// TwinCAT 3 PLC project PlcOpen_Test
// ProgramVersion: 3.1.4024.0
// libraries:
//   Tc2_Standard, * (Beckhoff Automation GmbH)
//   Tc2_System, * (Beckhoff Automation GmbH)
//   Tc2_Utilities, * (Beckhoff Automation GmbH)
//   Tc3_Module, * (Beckhoff Automation GmbH)
//   Tc3_PLCopen_OpcUa, * (Beckhoff Automation GmbH)
//   Tc2_OpcUa,3.3.2.0,Beckhoff Automation GmbH
// project tree:
//   DUTs/01_Strukturen/ SystemControlWord.TcDUT, SystemStatusWord.TcDUT
//   / GlobalTextList.TcGTLO, PlcTask.TcTTO, Visualisierungsmanager.TcVMO (not stored), VISU_TASK.TcTTO
//   GVLs/ GVL.TcGVL
//   POUs/01_Funktionsblock/ FB_Kommunikation.TcPOU
//   POUs/ Anlage.TcPOU, MAIN.TcPOU
//   VISUs/ Test_Visu.TcVIS
// real-time tasks:
//   TASK PlcTask: cycle T#10ms, priority 20, ADS port 350
//   TASK VISU_TASK: cycle T#200000us, priority 30, ADS port 351

CONFIGURATION PlcOpen_Test
    RESOURCE PLC ON TwinCAT3
        TASK PlcTask(INTERVAL := T#10ms, PRIORITY := 20);
        TASK VISU_TASK(INTERVAL := T#200000us, PRIORITY := 30);
        PROGRAM MAIN WITH PlcTask : MAIN;
        PROGRAM VisuElems_Visu_Prg WITH VISU_TASK : VisuElems.Visu_Prg;
    END_RESOURCE
END_CONFIGURATION

// ---- DUTs/01_Strukturen/SystemControlWord.TcDUT
TYPE SystemControlWord :
STRUCT			
	PowerOn			:BOOL;			// Einschalten von Reaktoreinheit
	SekReakt		:INT;			// Definierter sekundär-Reaktor
	Leitung			:INT;			// Definiert welche Leitung verwendet wird
	Temp			:REAL;			// Definierte Temperatur für Heiz- / Kühlprozess
	Enlteermenge	:REAL;			// Zu entleerende Menge
	Pumpmenge		:REAL;			// Zu pumpende Menge
	Haltedauer		:TIME;			// Wie lange soll TEmperatur gehalten werden
	Ruehrdauer		:TIME;			// Wie lange soll gerührt werden 
	Wartedauer		:TIME;			// Wie lange soll gerührt werden
	Zirkulierdauer	:TIME;			// Wie lange soll zirkuliert werden
END_STRUCT
END_TYPE

// ---- DUTs/01_Strukturen/SystemStatusWord.TcDUT
TYPE SystemStatusWord :
STRUCT
	SysReady		:BOOL;		// System ist eingeschalten und bereit
	PrimReady		:BOOL;		// Primärreaktor ist bereit für den Prozess
	PrimActiv		:BOOL;		// Primärreaktor führt Prozess aus
	SekReady		:BOOL;		// Sekundärreaktor ist bereit für den Prozess
	SekActiv		:BOOL;		// Sekundärreaktor führt Prozess aus
	GF1Activ		:BOOL;		// Heiz- / Kühlprozess läuft
	GF2Activ		:BOOL;		// Entleerprozess läuft
	GF3Activ		:BOOL;		// Pumpprozess läuft
	GF4Activ		:BOOL;		// Halteprozess läuft
	GF5Activ		:BOOL;		// Rührprozess läuft
	GF6Activ		:BOOL;		// Warteprozess läuft
	GF7Activ		:BOOL;		// Auffüllprozess läuft
	GF8Activ		:BOOL;		// Zirkulierprozess läuft
END_STRUCT
END_TYPE

// ---- GVLs/GVL.TcGVL
{attribute 'qualified_only'}
VAR_GLOBAL
	IP			:STRING(MAX_STRING_LENGTH) := 'opc.tcp://169.254.240.2:4840';
	NameSpace	:STRING(MAX_STRING_LENGTH) := 'urn:BeckhoffAutomation:Ua:PLC1';
	
	SW		:SystemStatusWord;
	CW		:SystemControlWord;
END_VAR

// ---- POUs/MAIN.TcPOU
PROGRAM MAIN
VAR
	Check			:BOOL;
END_VAR

Anlage();

END_PROGRAM

// ---- POUs/Anlage.TcPOU
PROGRAM Anlage
VAR
	Kom_Reaktor_1		:FB_Kommunikation;
	
END_VAR

Kom_Reaktor_1(I_sIP := GVL.IP, SW := GVL.SW); // FB_Kommunikation
GVL.CW := Kom_Reaktor_1.CW;

END_PROGRAM

// ---- POUs/01_Funktionsblock/FB_Kommunikation.TcPOU
FUNCTION_BLOCK FB_Kommunikation
VAR_INPUT
	I_sIP		:STRING;
	SW			:SystemStatusWord;
END_VAR

VAR_OUTPUT
	CW			:SystemControlWord;
	Busy		:BOOL;
	Error		:BOOL;
	ErrorID		:DWORD;
END_VAR

VAR
	Connect				:UA_Connect;
	Disconnect			:UA_Disconnect; 
	Read 				:UA_Read;
	Write				:UA_Write;
	Node				:UA_NodeGetHandle;
	NameSpaceIndex		:UA_GetNamespaceIndex;
	
	ConnectInfo			:ST_UASessionConnectInfo;
	NodeID				:ST_UANodeID;
	NodeInfo			:ST_UANodeAdditionalInfo;
	
	ConnectionHdl		:DWORD;
	NoteHdl				:DWORD;
	NameSpace			:UINT;
	IndexRangeCount		:UINT := 1;
	IndexRange			:ARRAY [1..nMaxIndexRange] OF ST_UAIndexRange;
	NodeIdentifier		:STRING(MAX_STRING_LENGTH) := 'GVL_OPC_UA.SW';
	ReadData			:SystemStatusWord; 		// change to node data type
END_VAR

// Definition der Verbindungsinformationen
ConnectInfo.tSessionTimeout := T#1M;
ConnectInfo.tConnectTimeout := T#1M;
ConnectInfo.sApplicationName := '';
ConnectInfo.eSecurityMode := eUASecurityMsgMode_Sign_Encrypt;				// 3 = Sign_Encrypted
ConnectInfo.eSecurityPolicyUri := eUASecurityPolicy_Basic256Sha256;			// 4 = Basic256  
ConnectInfo.eTransportProfileUri := eUATransportProfileUri_UATcp;			// 1 = UATcp
ConnectInfo.stUserIdentTokenType.eUserIdentTokenType := eUAUITT_Username;	// 1 = Username
ConnectInfo.stUserIdentTokenType.sTokenParam1 := 'Administrator';			// Username
ConnectInfo.stUserIdentTokenType.sTokenParam2 := '1';						// PW

GVL.SW := ReadData;

ACTION ACT_Connect:
Connect(ServerUrl := I_sIP, SessionConnectInfo := ConnectInfo, Timeout := T#5s); // UA_Connect
Busy := Connect.Busy;
ConnectionHdl := Connect.ConnectionHdl;
Error := Connect.Error;
ErrorID := Connect.ErrorID;
END_ACTION

ACTION ACT_Disconnect:
Busy := Disconnect.Busy;
Error := Disconnect.Error;
ErrorID := Disconnect.ErrorID;
Disconnect(ConnectionHdl := ConnectionHdl, Timeout := T#5s); // UA_Disconnect
END_ACTION

ACTION ACT_GetNameSpaceIndex:
Busy := NameSpaceIndex.Busy;
Error := NameSpaceIndex.Error;
ErrorID := NameSpaceIndex.ErrorID;
NameSpaceIndex(ConnectionHdl := ConnectionHdl, NamespaceUri := GVL.NameSpace, Timeout := T#5s); // UA_GetNamespaceIndex
NameSpace := NameSpaceIndex.NamespaceIndex;
END_ACTION

ACTION ACT_GetNodes:
NoteHdl := Node.NodeHdl;
Busy := Node.Busy;
Error := Node.Error;
ErrorID := Node.ErrorID;
Node(ConnectionHdl := ConnectionHdl, NodeID := NodeID, Timeout := T#5s); // UA_NodeGetHandle
END_ACTION

ACTION ACT_Read:
Busy := Read.Busy;
Error := Read.Error;
ErrorID := Read.ErrorID;
Read(
    ConnectionHdl := ConnectionHdl,
    NodeHdl := NoteHdl,
    stNodeAddInfo := NodeInfo,
    pVariable := ADR(ReadData),
    cbData := SIZEOF(ReadData),
    Timeout := T#5s); // UA_Read
END_ACTION

ACTION ACT_Write:
Write(); // UA_Write
END_ACTION

METHOD M_M_Connect : BOOL
VAR_INPUT
END_VAR
// Setzen der Ausführvariabel
Connect.Execute := TRUE;
// Aufrufen der Aktion
ACT_Connect();

// Methode abschliessen
IF Connect.Done THEN
	Connect.Execute := FALSE;
	M_M_Connect := TRUE;
END_IF
END_METHOD

METHOD M_M_Disconnect : BOOL
VAR_INPUT
END_VAR
// Setzen der Ausführvariabel
Disconnect.Execute := TRUE;
// Aufrufen der Aktion
Act_Disconnect();

// Methode abschliessen
IF Disconnect.Done THEN
	Disconnect.Execute := FALSE;
	M_M_Disconnect := TRUE;
END_IF
END_METHOD

METHOD M_M_GetNameSpaceIndex : BOOL
VAR_INPUT
END_VAR
// Setzen der Ausführvariabel
NameSpaceIndex.Execute := TRUE;
// Aufrufen der Aktion
ACT_GetNameSpaceIndex();

// Methode abschliessen
IF NameSpaceIndex.Done THEN
	NameSpaceIndex.Execute := FALSE;
	M_M_GetNameSpaceIndex := TRUE;
END_IF
END_METHOD

METHOD M_M_GetNodes : BOOL
VAR_INPUT
END_VAR
// Definieren von relevanten Parameter
NodeID.eIdentifierType := eUAIdentifierType_String;
NodeID.nNamespaceIndex := NameSpace;
NodeID.sIdentifier := NodeIdentifier;

// Setzen der Ausführvariabel
Node.Execute := TRUE;
// Aufrufen der Aktion
ACT_GetNodes();

// Methode abschliessen
IF Node.Done THEN
	Node.Execute := FALSE;
	M_M_getNodes := TRUE;
END_IF
END_METHOD

METHOD M_M_Read : BOOL
VAR_INPUT
END_VAR
// Definieren von Parametern
//NodeInfo.nIndexRangeCount := IndexRangeCount;
//NodeInfo.stIndexRange := IndexRange;

// Setzen der Ausführvariabel
Read.Execute := TRUE;
// Aufrufen der Aktion
ACT_Read();

// Methode abschliessen
IF Read.Done THEN
	Read.Execute := FALSE;
	M_M_Read := TRUE;
END_IF
END_METHOD

METHOD M_M_Write : BOOL
VAR_INPUT
END_VAR


// Methode abschliessen
IF Write.Done THEN
	Write.Execute := FALSE;
	M_M_Write := TRUE;
END_IF
END_METHOD

END_FUNCTION_BLOCK

// ---- GlobalTextList.TcGTLO
TEXTLIST GlobalTextList
  602 = '% %04x'
  213 = '%04x'
  132 = 'Busy:'
  727 = 'Connect'
  51 = 'Disconnect'
  925 = 'Error'
  519 = 'Error:'
  751 = 'Errorhandling'
  292 = 'ErrorID:'
  728 = 'GetNameSpaceIndex'
  678 = 'GetNotes'
  850 = 'Kommunikation'
  600 = 'Read'
END_TEXTLIST

// ---- VISUs/Test_Visu.TcVIS
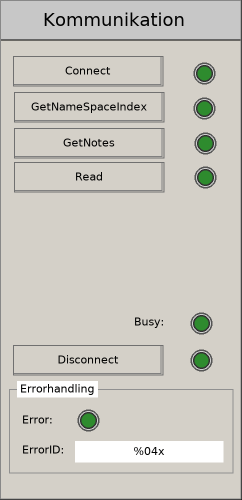
VISUALIZATION Test_Visu  // 242x500
    Rectangle (0,0 242x500)
    Rectangle (0,0 242x40)
    Label (39,5 150x30), "Kommunikation"
    GroupBox (9,381 224x92), "Errorhandling"
        Label (10,24 150x30), "Error:"
        Label (10,54 150x30), "ErrorID:"
        Lamp1 (67,27 25x25), variable: Anlage.Kom_Reaktor_1.Error, style: Lamp-Lamp1-Green
        Textfield (65,59 150x23), "%04x", text variable: Anlage.Kom_Reaktor_1.ErrorID, input disabled if: TRUE
    Button (13,56 150x30), "Connect"
        OnMouseClick: execute { Anlage.Kom_Reaktor_1.M_M_Connect(); }
    Button (14,92 150x30), "GetNameSpaceIndex"
        OnMouseClick: execute { Anlage.Kom_Reaktor_1.M_M_GetNameSpaceIndex(); }
    Button (14,128 150x30), "GetNotes"
        OnMouseClick: execute { Anlage.Kom_Reaktor_1.M_M_GetNodes(); }
    Button (14,162 150x30), "Read"
        OnMouseClick: execute { Anlage.Kom_Reaktor_1.M_M_Read(); }
    Button (13,345 150x30), "Disconnect"
        OnMouseClick: execute { Anlage.Kom_Reaktor_1.M_M_Disconnect(); }
    Lamp1 (192,61 25x25), variable: Anlage.Kom_Reaktor_1.Connect.Done, style: Lamp-Lamp1-Green
    Lamp1 (192,96 25x25), variable: Anlage.Kom_Reaktor_1.NameSpaceIndex.Done, style: Lamp-Lamp1-Green
    Lamp1 (193,131 25x25), variable: Anlage.Kom_Reaktor_1.Node.Done, style: Lamp-Lamp1-Green
    Lamp1 (193,165 25x25), variable: Anlage.Kom_Reaktor_1.Read.Done, style: Lamp-Lamp1-Green
    Lamp1 (189,348 25x25), variable: Anlage.Kom_Reaktor_1.Disconnect.Done, style: Lamp-Lamp1-Green
    Lamp1 (189,311 25x25), variable: Anlage.Kom_Reaktor_1.Busy, style: Lamp-Lamp1-Green
    Label (131,307 44x30), "Busy:"
END_VISUALIZATION
